FUNCTION MULTIME
  (* Standard: 61499-1 *)
  (* Version 1.0, 2025-12-21, Franz Höpfinger *)
  PACKAGE OSCAT::Basic::POUs::Time_Date;
  IMPORT eclipse4diac::core::TypeHash;
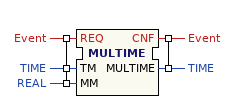
  EVENT_INPUT
    REQ WITH TM, MM;
  END_EVENT
  EVENT_OUTPUT
    CNF WITH MULTIME;
  END_EVENT
  VAR_INPUT
    TM : TIME;
    MM : REAL;
  END_VAR
  VAR_OUTPUT
    MULTIME : TIME;
  END_VAR
  BODY IN ST:
PACKAGE OSCAT::Basic::POUs::Time_Date;

FUNCTION MULTIME : TIME
VAR_INPUT
	TM : TIME;
	MM : REAL;
END_VAR

(*
 * version 1.1	14 mar 2008 programmer 	hugo tested by		tobias
 * *
 * multiplies a time by a real number and returns a time
 *)
MULTIME := TM * MM;

END_FUNCTION
(* revision history hm		2. oct 2006	rev 1.0 original version
 * *
 * hm		14. mar 2008	rev 1.1 rounded the result after the last digit *)
  END_BODY
END_FUNCTION
